(* CoDeSys 2.3 export: NETVARDATAITEM_UDP.EXP *)

(* Data type *)
TYPE NetVarDataItem_Udp :
STRUCT
	pAdress		: POINTER TO ARRAY[0..255] OF BYTE;
	nDataLen	: NetVarDataLen_Udp;
END_STRUCT
END_TYPE
